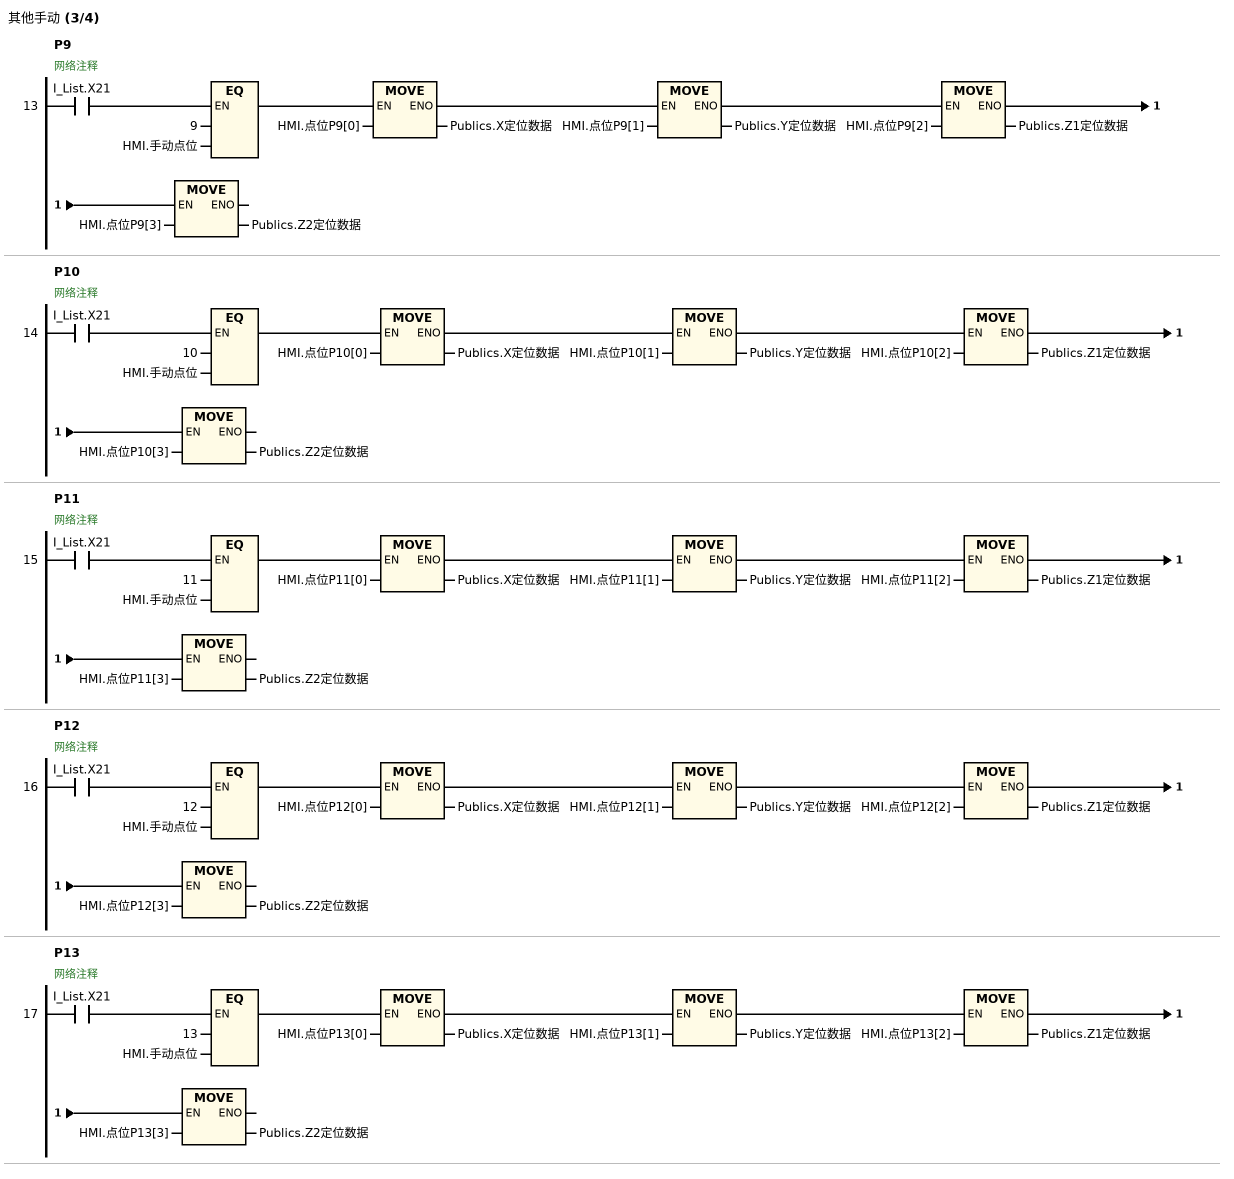
// NETWORK 13: P9
// 网络注释
_w9 := I_List.X21 AND 9 = HMI.手动点位;
IF _w9 THEN Publics.X定位数据 := HMI.点位P9[0]; END_IF
IF _w9 THEN Publics.Y定位数据 := HMI.点位P9[1]; END_IF
IF _w9 THEN Publics.Z1定位数据 := HMI.点位P9[2]; END_IF
IF _w9 THEN Publics.Z2定位数据 := HMI.点位P9[3]; END_IF

// NETWORK 14: P10
// 网络注释
_w10 := I_List.X21 AND 10 = HMI.手动点位;
IF _w10 THEN Publics.X定位数据 := HMI.点位P10[0]; END_IF
IF _w10 THEN Publics.Y定位数据 := HMI.点位P10[1]; END_IF
IF _w10 THEN Publics.Z1定位数据 := HMI.点位P10[2]; END_IF
IF _w10 THEN Publics.Z2定位数据 := HMI.点位P10[3]; END_IF

// NETWORK 15: P11
// 网络注释
_w11 := I_List.X21 AND 11 = HMI.手动点位;
IF _w11 THEN Publics.X定位数据 := HMI.点位P11[0]; END_IF
IF _w11 THEN Publics.Y定位数据 := HMI.点位P11[1]; END_IF
IF _w11 THEN Publics.Z1定位数据 := HMI.点位P11[2]; END_IF
IF _w11 THEN Publics.Z2定位数据 := HMI.点位P11[3]; END_IF

// NETWORK 16: P12
// 网络注释
_w12 := I_List.X21 AND 12 = HMI.手动点位;
IF _w12 THEN Publics.X定位数据 := HMI.点位P12[0]; END_IF
IF _w12 THEN Publics.Y定位数据 := HMI.点位P12[1]; END_IF
IF _w12 THEN Publics.Z1定位数据 := HMI.点位P12[2]; END_IF
IF _w12 THEN Publics.Z2定位数据 := HMI.点位P12[3]; END_IF

// NETWORK 17: P13
// 网络注释
_w13 := I_List.X21 AND 13 = HMI.手动点位;
IF _w13 THEN Publics.X定位数据 := HMI.点位P13[0]; END_IF
IF _w13 THEN Publics.Y定位数据 := HMI.点位P13[1]; END_IF
IF _w13 THEN Publics.Z1定位数据 := HMI.点位P13[2]; END_IF
IF _w13 THEN Publics.Z2定位数据 := HMI.点位P13[3]; END_IF

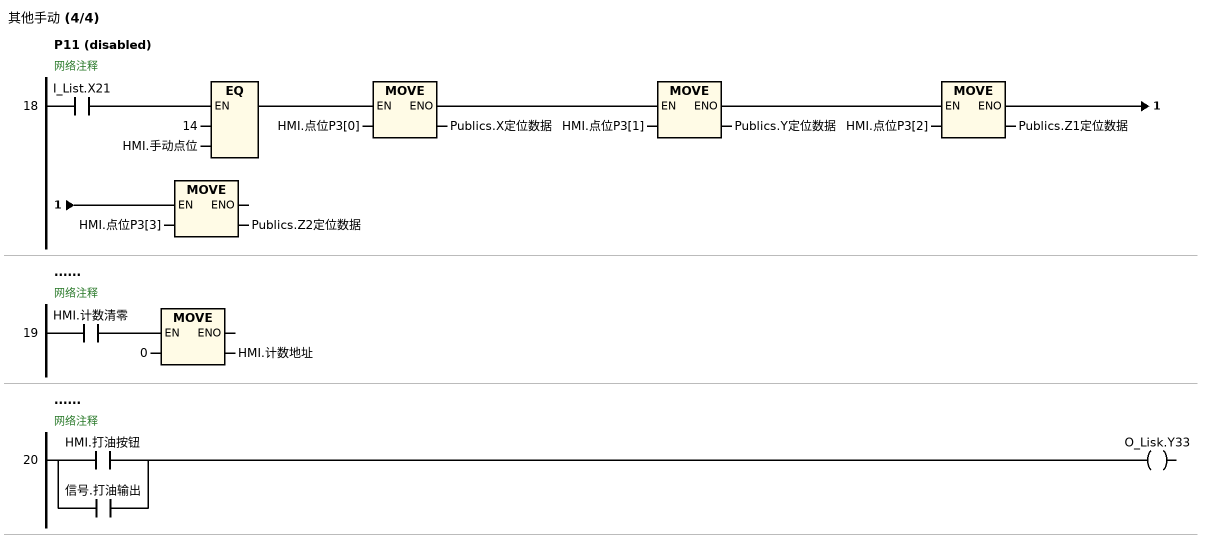
// NETWORK 18: P11 (disabled)
// 网络注释
// _w14 := I_List.X21 AND 14 = HMI.手动点位;
// IF _w14 THEN Publics.X定位数据 := HMI.点位P3[0]; END_IF
// IF _w14 THEN Publics.Y定位数据 := HMI.点位P3[1]; END_IF
// IF _w14 THEN Publics.Z1定位数据 := HMI.点位P3[2]; END_IF
// IF _w14 THEN Publics.Z2定位数据 := HMI.点位P3[3]; END_IF

// NETWORK 19: ......
// 网络注释
IF HMI.计数清零 THEN HMI.计数地址 := 0; END_IF

// NETWORK 20: ......
// 网络注释
O_Lisk.Y33 := HMI.打油按钮 OR 信号.打油输出;

END_PROGRAM

// Device/Application/Servo_Ctrol
PROGRAM Servo_Ctrol
VAR
	总线复位: BOOL;
	SMC3_ReinitDrive_0: SMC3_ReinitDrive;
	SMC3_ReinitDrive_1: SMC3_ReinitDrive;
	SMC3_ReinitDrive_2: SMC3_ReinitDrive;
	SMC3_ReinitDrive_3: SMC3_ReinitDrive;
	Y轴_使能: MC_Power;
	Z2轴_使能: MC_Power;
	Z1轴_使能: MC_Power;
	X轴_使能: MC_Power;
	MC_Jog_0: MC_Jog;
	Y轴_JOG: MC_Jog;
	Z2轴_JOG: MC_Jog;
	Z1轴_JOG: MC_Jog;
	X轴_JOG: MC_Jog;
	AXIS3: AXIS_REF_SM3;
	MC_Reset_0: MC_Reset;
	MC_Reset_1: MC_Reset;
	MC_Reset_2: MC_Reset;
	MC_Reset_3: MC_Reset;
	MC_ReadStatus_0: MC_ReadStatus;
	MC_ReadAxisError_0: MC_ReadAxisError;
	MC_ReadActualPosition_0: MC_ReadActualPosition;
	MC_ReadActualPosition_1: MC_ReadActualPosition;
	MC_ReadActualPosition_2: MC_ReadActualPosition;
	MC_ReadActualPosition_3: MC_ReadActualPosition;
	MC_Halt_0: MC_Halt;
	MC_Halt_1: MC_Halt;
	MC_Halt_2: MC_Halt;
	MC_Halt_3: MC_Halt;
	MC_Stop_0: MC_Stop;
	MC_Stop_1: MC_Stop;
	MC_Stop_2: MC_Stop;
	MC_Stop_3: MC_Stop;
	Z2定位: MC_MoveAbsolute;
	Z1定位: MC_MoveAbsolute;
	Y定位: MC_MoveAbsolute;
	X定位: MC_MoveAbsolute;
	MC_Home_0: MC_Home;
	MC_Home_1: MC_Home;
	MC_Home_2: MC_Home;
	MC_Home_3: MC_Home;
	ALM0: BOOL;
	ALM1: BOOL;
	ALM2: BOOL;
	ALM3: BOOL;
END_VAR
VAR // added by the converter: edge detectors and wires of the graphical bodies
    _rt1, _rt2, _rt3, _rt4, _rt5, _rt6, _rt7 : R_TRIG;
END_VAR

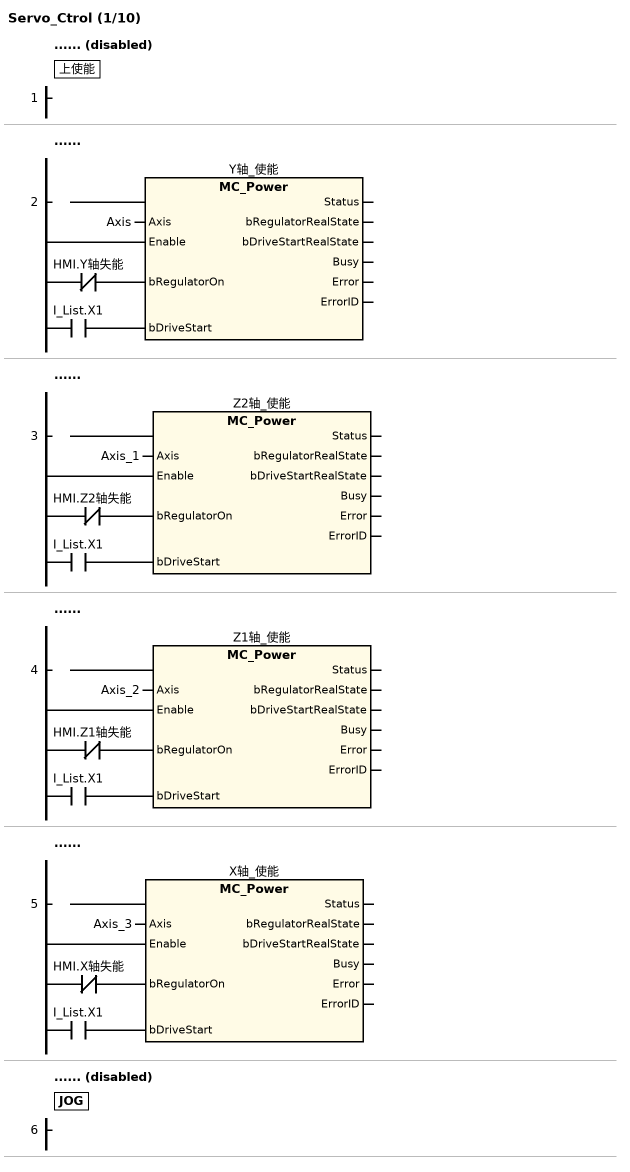
// NETWORK 1: ...... (disabled)
// label: 上使能

// NETWORK 2: ......
Y轴_使能(Axis := Axis, Enable := TRUE, bRegulatorOn := NOT HMI.Y轴失能, bDriveStart := I_List.X1); // MC_Power

// NETWORK 3: ......
Z2轴_使能(Axis := Axis_1, Enable := TRUE, bRegulatorOn := NOT HMI.Z2轴失能, bDriveStart := I_List.X1); // MC_Power

// NETWORK 4: ......
Z1轴_使能(Axis := Axis_2, Enable := TRUE, bRegulatorOn := NOT HMI.Z1轴失能, bDriveStart := I_List.X1); // MC_Power

// NETWORK 5: ......
X轴_使能(Axis := Axis_3, Enable := TRUE, bRegulatorOn := NOT HMI.X轴失能, bDriveStart := I_List.X1); // MC_Power

// NETWORK 6: ...... (disabled)
// label: JOG

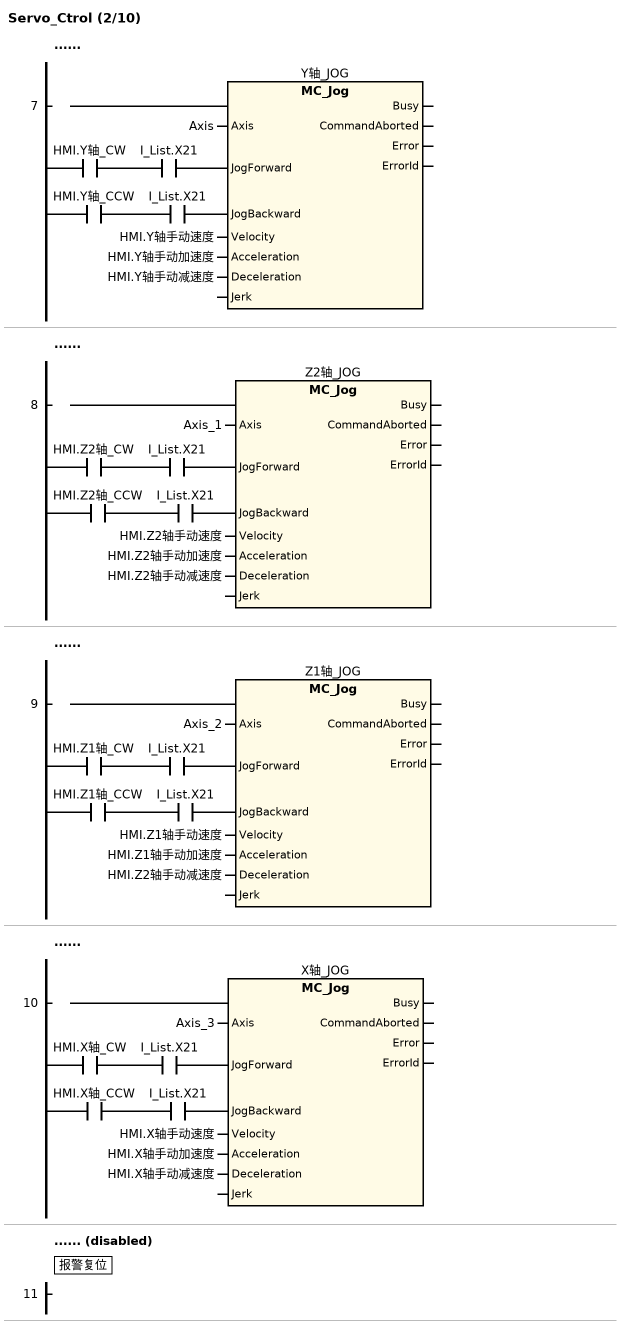
// NETWORK 7: ......
Y轴_JOG(
    Axis := Axis,
    JogForward := HMI.Y轴_CW AND I_List.X21,
    JogBackward := HMI.Y轴_CCW AND I_List.X21,
    Velocity := HMI.Y轴手动速度,
    Acceleration := HMI.Y轴手动加速度,
    Deceleration := HMI.Y轴手动减速度); // MC_Jog

// NETWORK 8: ......
Z2轴_JOG(
    Axis := Axis_1,
    JogForward := HMI.Z2轴_CW AND I_List.X21,
    JogBackward := HMI.Z2轴_CCW AND I_List.X21,
    Velocity := HMI.Z2轴手动速度,
    Acceleration := HMI.Z2轴手动加速度,
    Deceleration := HMI.Z2轴手动减速度); // MC_Jog

// NETWORK 9: ......
Z1轴_JOG(
    Axis := Axis_2,
    JogForward := HMI.Z1轴_CW AND I_List.X21,
    JogBackward := HMI.Z1轴_CCW AND I_List.X21,
    Velocity := HMI.Z1轴手动速度,
    Acceleration := HMI.Z1轴手动加速度,
    Deceleration := HMI.Z2轴手动减速度); // MC_Jog

// NETWORK 10: ......
X轴_JOG(
    Axis := Axis_3,
    JogForward := HMI.X轴_CW AND I_List.X21,
    JogBackward := HMI.X轴_CCW AND I_List.X21,
    Velocity := HMI.X轴手动速度,
    Acceleration := HMI.X轴手动加速度,
    Deceleration := HMI.X轴手动减速度); // MC_Jog

// NETWORK 11: ...... (disabled)
// label: 报警复位

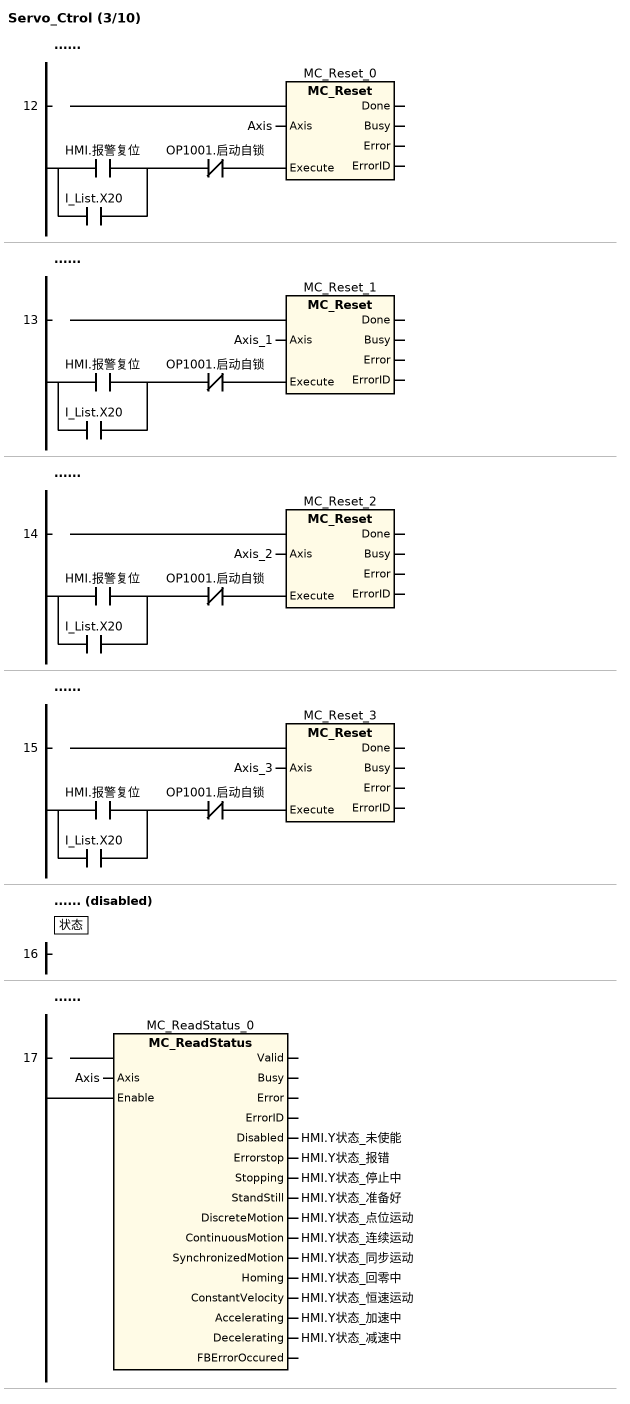
// NETWORK 12: ......
MC_Reset_0(Axis := Axis, Execute := (HMI.报警复位 OR I_List.X20) AND NOT OP1001.启动自锁); // MC_Reset

// NETWORK 13: ......
MC_Reset_1(Axis := Axis_1, Execute := (HMI.报警复位 OR I_List.X20) AND NOT OP1001.启动自锁); // MC_Reset

// NETWORK 14: ......
MC_Reset_2(Axis := Axis_2, Execute := (HMI.报警复位 OR I_List.X20) AND NOT OP1001.启动自锁); // MC_Reset

// NETWORK 15: ......
MC_Reset_3(Axis := Axis_3, Execute := (HMI.报警复位 OR I_List.X20) AND NOT OP1001.启动自锁); // MC_Reset

// NETWORK 16: ...... (disabled)
// label: 状态

// NETWORK 17: ......
MC_ReadStatus_0(
    Axis := Axis,
    Enable := TRUE,
    Disabled => HMI.Y状态_未使能,
    Errorstop => HMI.Y状态_报错,
    Stopping => HMI.Y状态_停止中,
    StandStill => HMI.Y状态_准备好,
    DiscreteMotion => HMI.Y状态_点位运动,
    ContinuousMotion => HMI.Y状态_连续运动,
    SynchronizedMotion => HMI.Y状态_同步运动,
    Homing => HMI.Y状态_回零中,
    ConstantVelocity => HMI.Y状态_恒速运动,
    Accelerating => HMI.Y状态_加速中,
    Decelerating => HMI.Y状态_减速中); // MC_ReadStatus

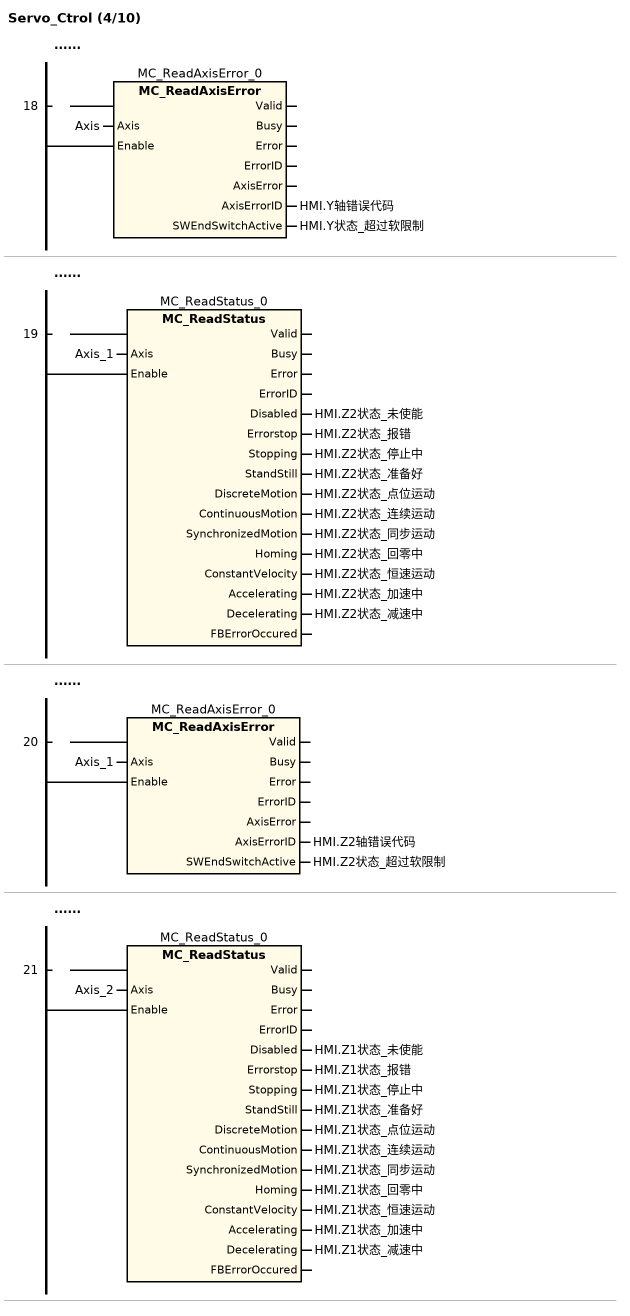
// NETWORK 18: ......
MC_ReadAxisError_0(
    Axis := Axis,
    Enable := TRUE,
    AxisErrorID => HMI.Y轴错误代码,
    SWEndSwitchActive => HMI.Y状态_超过软限制); // MC_ReadAxisError

// NETWORK 19: ......
MC_ReadStatus_0(
    Axis := Axis_1,
    Enable := TRUE,
    Disabled => HMI.Z2状态_未使能,
    Errorstop => HMI.Z2状态_报错,
    Stopping => HMI.Z2状态_停止中,
    StandStill => HMI.Z2状态_准备好,
    DiscreteMotion => HMI.Z2状态_点位运动,
    ContinuousMotion => HMI.Z2状态_连续运动,
    SynchronizedMotion => HMI.Z2状态_同步运动,
    Homing => HMI.Z2状态_回零中,
    ConstantVelocity => HMI.Z2状态_恒速运动,
    Accelerating => HMI.Z2状态_加速中,
    Decelerating => HMI.Z2状态_减速中); // MC_ReadStatus

// NETWORK 20: ......
MC_ReadAxisError_0(
    Axis := Axis_1,
    Enable := TRUE,
    AxisErrorID => HMI.Z2轴错误代码,
    SWEndSwitchActive => HMI.Z2状态_超过软限制); // MC_ReadAxisError

// NETWORK 21: ......
MC_ReadStatus_0(
    Axis := Axis_2,
    Enable := TRUE,
    Disabled => HMI.Z1状态_未使能,
    Errorstop => HMI.Z1状态_报错,
    Stopping => HMI.Z1状态_停止中,
    StandStill => HMI.Z1状态_准备好,
    DiscreteMotion => HMI.Z1状态_点位运动,
    ContinuousMotion => HMI.Z1状态_连续运动,
    SynchronizedMotion => HMI.Z1状态_同步运动,
    Homing => HMI.Z1状态_回零中,
    ConstantVelocity => HMI.Z1状态_恒速运动,
    Accelerating => HMI.Z1状态_加速中,
    Decelerating => HMI.Z1状态_减速中); // MC_ReadStatus

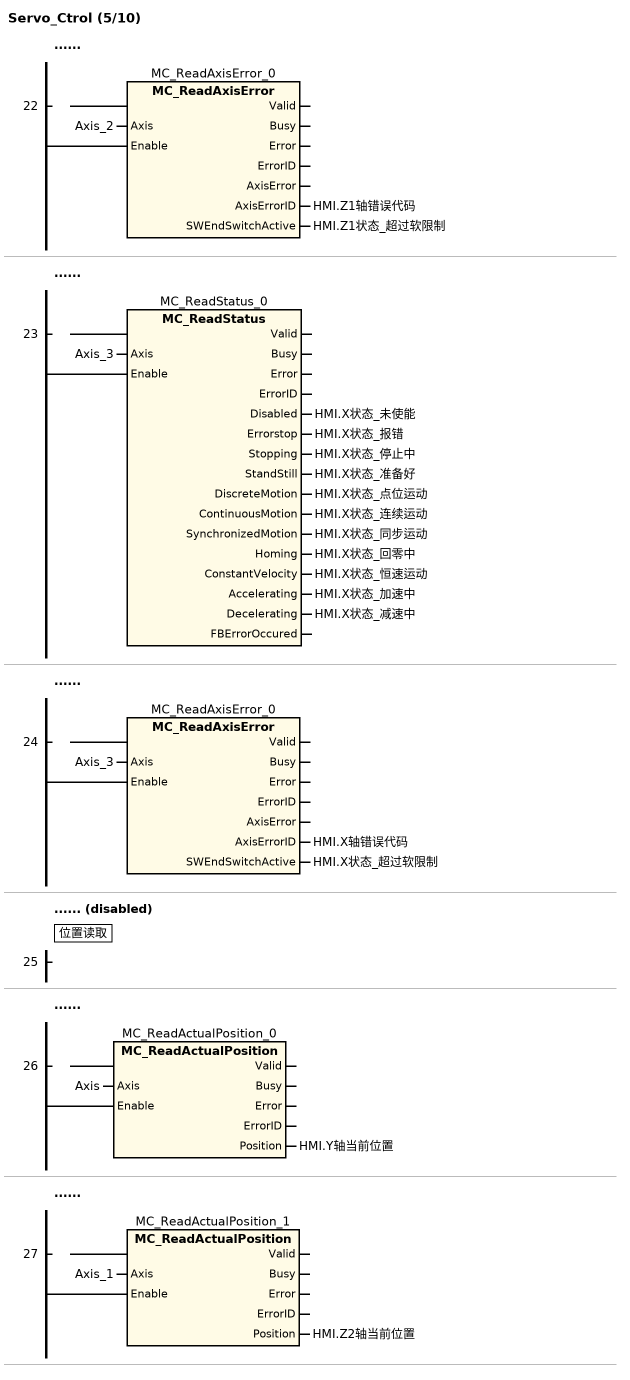
// NETWORK 22: ......
MC_ReadAxisError_0(
    Axis := Axis_2,
    Enable := TRUE,
    AxisErrorID => HMI.Z1轴错误代码,
    SWEndSwitchActive => HMI.Z1状态_超过软限制); // MC_ReadAxisError

// NETWORK 23: ......
MC_ReadStatus_0(
    Axis := Axis_3,
    Enable := TRUE,
    Disabled => HMI.X状态_未使能,
    Errorstop => HMI.X状态_报错,
    Stopping => HMI.X状态_停止中,
    StandStill => HMI.X状态_准备好,
    DiscreteMotion => HMI.X状态_点位运动,
    ContinuousMotion => HMI.X状态_连续运动,
    SynchronizedMotion => HMI.X状态_同步运动,
    Homing => HMI.X状态_回零中,
    ConstantVelocity => HMI.X状态_恒速运动,
    Accelerating => HMI.X状态_加速中,
    Decelerating => HMI.X状态_减速中); // MC_ReadStatus

// NETWORK 24: ......
MC_ReadAxisError_0(
    Axis := Axis_3,
    Enable := TRUE,
    AxisErrorID => HMI.X轴错误代码,
    SWEndSwitchActive => HMI.X状态_超过软限制); // MC_ReadAxisError

// NETWORK 25: ...... (disabled)
// label: 位置读取

// NETWORK 26: ......
MC_ReadActualPosition_0(Axis := Axis, Enable := TRUE, Position => HMI.Y轴当前位置); // MC_ReadActualPosition

// NETWORK 27: ......
MC_ReadActualPosition_1(Axis := Axis_1, Enable := TRUE, Position => HMI.Z2轴当前位置); // MC_ReadActualPosition

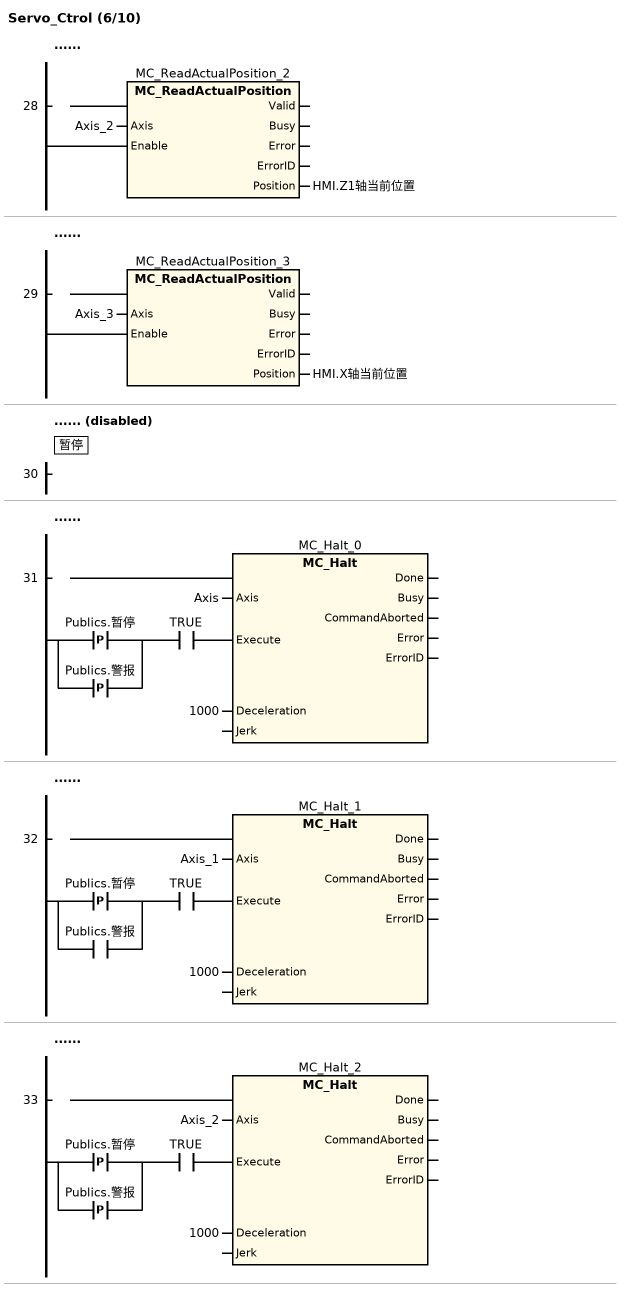
// NETWORK 28: ......
MC_ReadActualPosition_2(Axis := Axis_2, Enable := TRUE, Position => HMI.Z1轴当前位置); // MC_ReadActualPosition

// NETWORK 29: ......
MC_ReadActualPosition_3(Axis := Axis_3, Enable := TRUE, Position => HMI.X轴当前位置); // MC_ReadActualPosition

// NETWORK 30: ...... (disabled)
// label: 暂停

// NETWORK 31: ......
_rt1(CLK := Publics.暂停);
_rt2(CLK := Publics.警报);
MC_Halt_0(Axis := Axis, Execute := (_rt1.Q OR _rt2.Q) AND TRUE, Deceleration := 1000); // MC_Halt

// NETWORK 32: ......
_rt3(CLK := Publics.暂停);
MC_Halt_1(Axis := Axis_1, Execute := (_rt3.Q OR Publics.警报) AND TRUE, Deceleration := 1000); // MC_Halt

// NETWORK 33: ......
_rt4(CLK := Publics.暂停);
_rt5(CLK := Publics.警报);
MC_Halt_2(Axis := Axis_2, Execute := (_rt4.Q OR _rt5.Q) AND TRUE, Deceleration := 1000); // MC_Halt

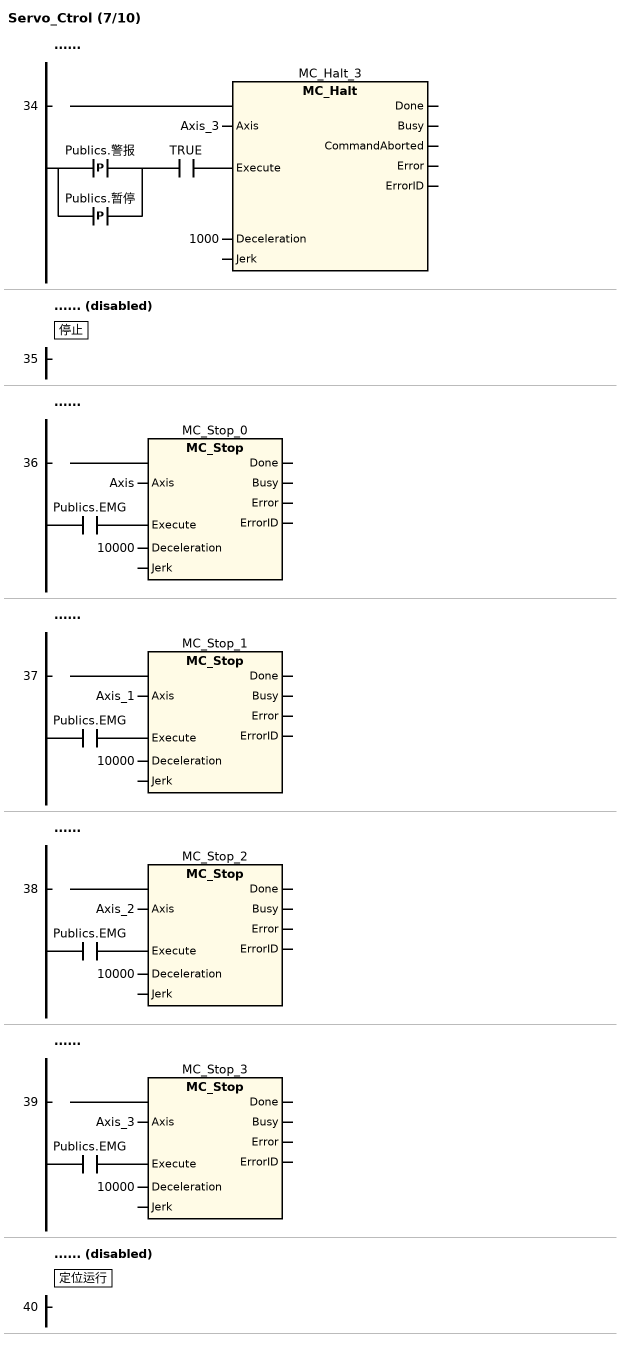
// NETWORK 34: ......
_rt6(CLK := Publics.警报);
_rt7(CLK := Publics.暂停);
MC_Halt_3(Axis := Axis_3, Execute := (_rt6.Q OR _rt7.Q) AND TRUE, Deceleration := 1000); // MC_Halt

// NETWORK 35: ...... (disabled)
// label: 停止

// NETWORK 36: ......
MC_Stop_0(Axis := Axis, Execute := Publics.EMG, Deceleration := 10000); // MC_Stop

// NETWORK 37: ......
MC_Stop_1(Axis := Axis_1, Execute := Publics.EMG, Deceleration := 10000); // MC_Stop

// NETWORK 38: ......
MC_Stop_2(Axis := Axis_2, Execute := Publics.EMG, Deceleration := 10000); // MC_Stop

// NETWORK 39: ......
MC_Stop_3(Axis := Axis_3, Execute := Publics.EMG, Deceleration := 10000); // MC_Stop

// NETWORK 40: ...... (disabled)
// label: 定位运行

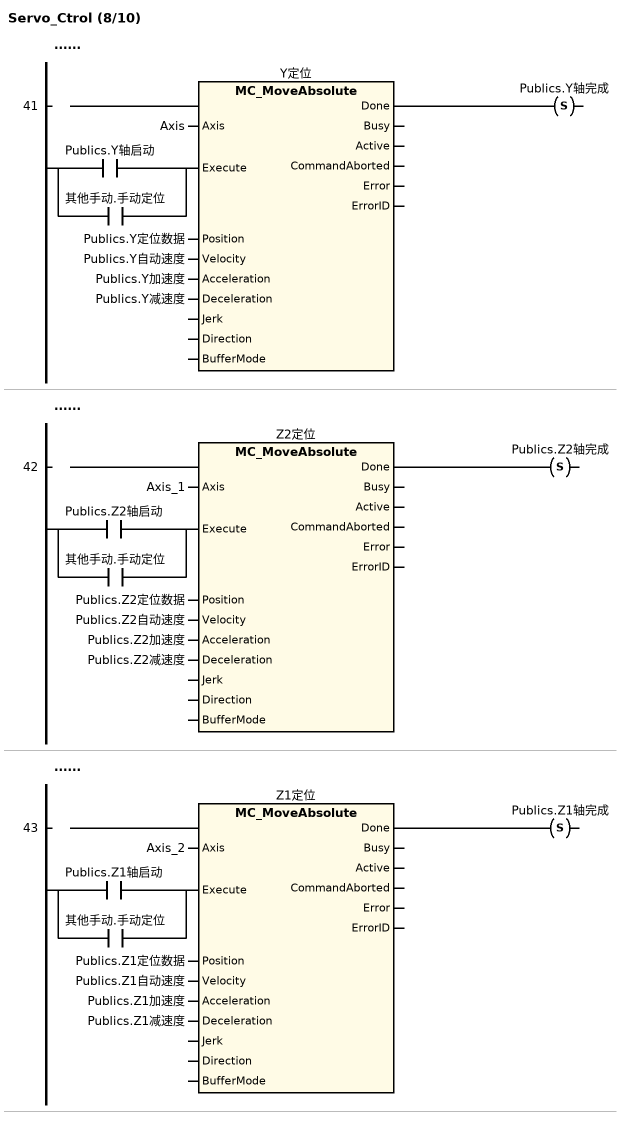
// NETWORK 41: ......
Y定位(
    Axis := Axis,
    Execute := Publics.Y轴启动 OR 其他手动.手动定位,
    Position := Publics.Y定位数据,
    Velocity := Publics.Y自动速度,
    Acceleration := Publics.Y加速度,
    Deceleration := Publics.Y减速度); // MC_MoveAbsolute
Publics.Y轴完成 S= Y定位.Done;

// NETWORK 42: ......
Z2定位(
    Axis := Axis_1,
    Execute := Publics.Z2轴启动 OR 其他手动.手动定位,
    Position := Publics.Z2定位数据,
    Velocity := Publics.Z2自动速度,
    Acceleration := Publics.Z2加速度,
    Deceleration := Publics.Z2减速度); // MC_MoveAbsolute
Publics.Z2轴完成 S= Z2定位.Done;

// NETWORK 43: ......
Z1定位(
    Axis := Axis_2,
    Execute := Publics.Z1轴启动 OR 其他手动.手动定位,
    Position := Publics.Z1定位数据,
    Velocity := Publics.Z1自动速度,
    Acceleration := Publics.Z1加速度,
    Deceleration := Publics.Z1减速度); // MC_MoveAbsolute
Publics.Z1轴完成 S= Z1定位.Done;

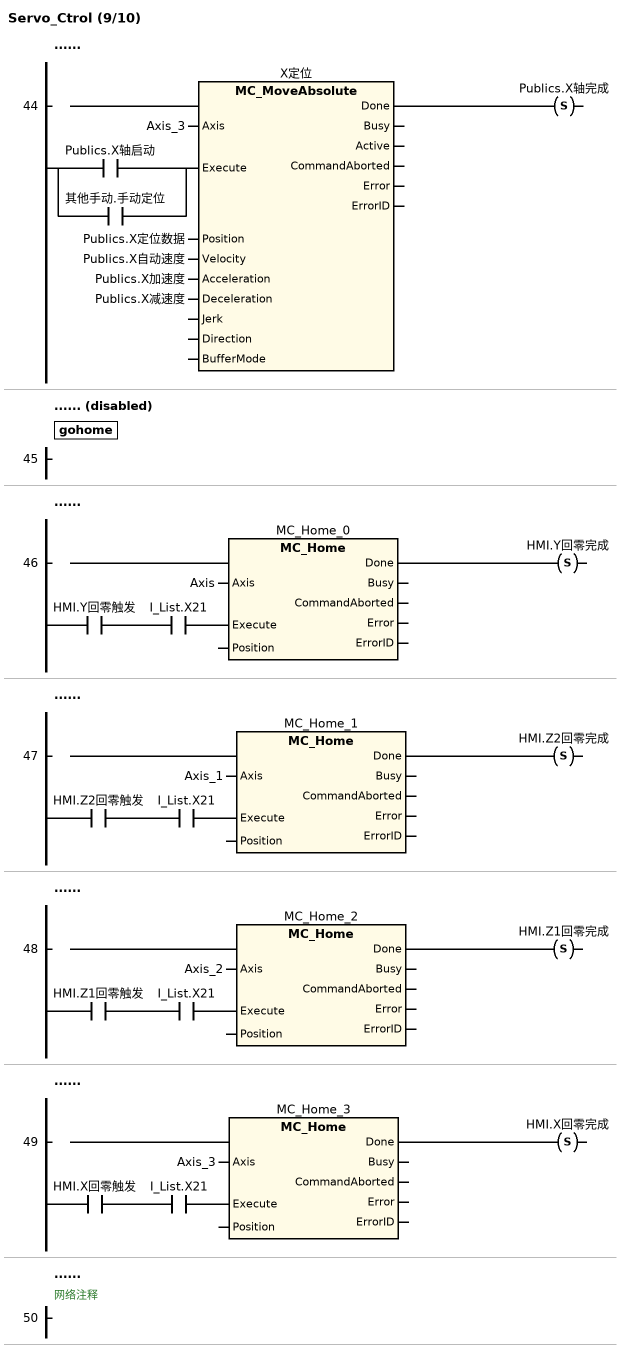
// NETWORK 44: ......
X定位(
    Axis := Axis_3,
    Execute := Publics.X轴启动 OR 其他手动.手动定位,
    Position := Publics.X定位数据,
    Velocity := Publics.X自动速度,
    Acceleration := Publics.X加速度,
    Deceleration := Publics.X减速度); // MC_MoveAbsolute
Publics.X轴完成 S= X定位.Done;

// NETWORK 45: ...... (disabled)
// label: gohome

// NETWORK 46: ......
MC_Home_0(Axis := Axis, Execute := HMI.Y回零触发 AND I_List.X21); // MC_Home
HMI.Y回零完成 S= MC_Home_0.Done;

// NETWORK 47: ......
MC_Home_1(Axis := Axis_1, Execute := HMI.Z2回零触发 AND I_List.X21); // MC_Home
HMI.Z2回零完成 S= MC_Home_1.Done;

// NETWORK 48: ......
MC_Home_2(Axis := Axis_2, Execute := HMI.Z1回零触发 AND I_List.X21); // MC_Home
HMI.Z1回零完成 S= MC_Home_2.Done;

// NETWORK 49: ......
MC_Home_3(Axis := Axis_3, Execute := HMI.X回零触发 AND I_List.X21); // MC_Home
HMI.X回零完成 S= MC_Home_3.Done;

// NETWORK 50: ......
// 网络注释

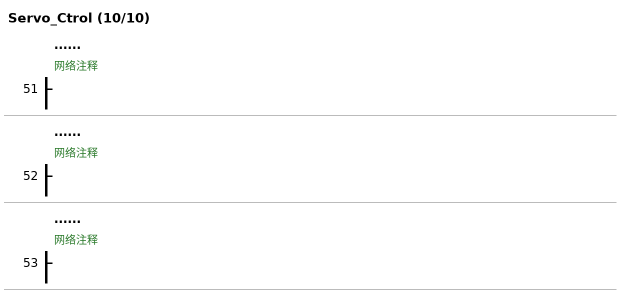
// NETWORK 51: ......
// 网络注释

// NETWORK 52: ......
// 网络注释

// NETWORK 53: ......
// 网络注释

END_PROGRAM

// Device/Application/ITF
INTERFACE ITF

END_INTERFACE

// Device/Application/FunctionBlock/FB_CylinderDouble
FUNCTION_BLOCK FB_CylinderDouble
VAR_IN_OUT
	///气缸控制、状态和报警
	stCylvar: CYLINDER_REF;
END_VAR
VAR_INPUT
	///安全条件
	xReady: BOOL;
	///报警复位
	xReset: BOOL;
	///手动控制,每on一次,则反转输出点状态
	xManuCmd: BOOL;
	///原位检测
	xBackSensor: BOOL;
	///到位检测
	xFrontSensor: BOOL;
	///手自动不一致报警无效
	xManuAlmDisable: BOOL;
	///原位检测无效
	xBackSensorDisable: BOOL;
	///到位检测无效	
	xFrontSensorDisable: BOOL;
	///原位延时	
	wBackDelay: WORD;
	///到位延时
	wFrontDelay: WORD;
END_VAR
VAR_OUTPUT
	///输出点,对应双控气缸原位电磁阀
	xOutputA: BOOL;
	///输出点,应双控气缸到位电磁阀
	xOutputB: BOOL;
	///未满足安全条件报警
	f_xNotRdyAlm: BOOL;
	///手自动不一致报警	
	f_xManuAlm: BOOL;
	///未在原位报警
	f_xBackAlm: BOOL;
	///未到位报警	
	f_xFrontAlm: BOOL;
	///气缸处于不受控制状态报警
	f_xUncontrolledAlm: BOOL;
END_VAR
VAR
	///获取自动控制的上升沿
	fbAutoRise: R_TRIG;
	///获取自动控制的下升沿
	fbAutoFall: F_TRIG;
	///获取手动控制的下升沿
	fbManuFall: F_TRIG;
	///获取复位信号的上升沿
	fbResetRise: R_TRIG;
	///原位状态延时,用于输出原位状态
	fbBackTon: TON;
	///到位状态延时,用于输出到位状态	
	fbFrontTon: TON;
	///获取原位状态下降沿
	fbBackFall: F_TRIG;
	///获取到位状态下降沿
	fbFrontFall: F_TRIG;
	///原位动作超时,用于输出未在原位位置报警
	fbBackWait: TON;
	///到位动作超时,用于输出未在原位位置报警
	fbFrontWait: TON;
END_VAR

   //初始化时返回原位
   IF  xReady AND stCylvar.xInit AND ( NOT xManuCmd ) THEN
	     xOutputA  := TRUE; 
         xOutputB  := FALSE;
		 f_xManuAlm  := FALSE;
		 stCylvar.xInit  := FALSE;	  	  	 	  
   END_IF	  
   
   //获取手动控制、自动控制的边沿信号
   fbManuFall(CLK:=xManuCmd , Q=> );
   fbAutoRise(CLK:=stCylvar.xAutoCmd , Q=> );
   fbAutoFall(CLK:=stCylvar.xAutoCmd , Q=> );
   
   //1,手动操作时，如果满足安全条件且未屏蔽手自动不一致报警时，则输出点A反转，输出点B取输出点A的反逻辑
   IF xReady AND (NOT xManuAlmDisable) AND fbManuFall.Q THEN
	   xOutputA  := NOT xOutputA; 
	   xOutputB  := NOT xOutputA;
	   
	//手动操作生效时，判断输出点状态与自动命令是否一致，不一致时,置位手动操作执行中报警；一致时复位该报警。
	//当因安全条件不满足导致自动命令未执行时，可通过手动操作控制其动作执行,此时手动操作并不引起手动操作执行中报警。
   	   IF (stCylvar.xAutoCmd AND (NOT xManuAlmDisable) ) XOR xOutputB THEN
   	   	    f_xManuAlm  :=TRUE;
   	   ELSE 
   	   	    f_xManuAlm  :=FALSE;
   	   END_IF
   END_IF
   //2,手动操作时，如果满足安全条件且屏蔽了手自动不一致报警时，则自动控制点反转、复位手自动不一致报警，  
    IF xReady AND  xManuAlmDisable AND fbManuFall.Q THEN
   	    stCylvar.xAutoCmd  := NOT stCylvar.xAutoCmd ;
		f_xManuAlm  :=FALSE;		  	 	
    END_IF
   
   //自动命令置位时，如满足安全条件，则输出点A复位、 输出点B置位。
   IF xReady AND fbAutoRise.Q THEN
   	    xOutputA  :=FALSE;
		xOutputB  :=TRUE;
		
   END_IF
   //自动命令复位时，如满足安全条件，则输出点A置位、 输出点B复位。
   IF xReady AND fbAutoFall.Q THEN
   	    xOutputA  :=TRUE;
		xOutputB  :=FALSE;		
   END_IF
   
   
   //到位状态输出
   fbFrontTon(IN:=( NOT xOutputA ) AND xOutputB AND ( xFrontSensor OR xFrontSensorDisable ) AND ( NOT xBackSensor ) , PT:= WORD_TO_TIME ( wFrontDelay *10 ), Q=> stCylvar.xIsFront, ET=> );
   
   //原位状态输出
   fbBackTon(IN:= xOutputA  AND ( NOT xOutputB) AND ( NOT xFrontSensor ) AND ( xBackSensor OR xBackSensorDisable ) , PT:= WORD_TO_TIME ( wBackDelay *10 ) , Q=> stCylvar.xIsBack, ET=> );
   
   
   //报警复位
   fbResetRise(CLK:= xReset, Q=> );
   IF fbResetRise.Q THEN
   	   f_xNotRdyAlm := FALSE;
	   f_xFrontAlm := FALSE;
	   f_xBackAlm := FALSE;
	   f_xUncontrolledAlm := FALSE;
   
   END_IF
   
   
   //未满足安全条件报警
   //当手动操作或自动命令状态发生改变时，如果不能满足安全条件，则输出未满足安全条件报警
   IF ( fbManuFall.Q OR fbAutoRise.Q OR fbAutoFall.Q ) AND ( NOT xReady ) THEN
   	   f_xNotRdyAlm := TRUE; 
   END_IF
   
   
   //未在原位报警
   //自动命令变OFF后(上电后气缸处于自由状态时不判断)，延时5秒，如果原位标志未变为ON、且未发生手动操作和安全条件报警，则输出未到原位报警
   fbBackWait(IN:= ( NOT stCylvar.xAutoCmd ) AND ( xOutputA OR xOutputB ) , PT:= T#5S , Q=> , ET=> );
   fbBackFall(CLK:= stCylvar.xIsBack , Q=> );
   IF (( fbBackWait.Q AND (NOT stCylvar.xIsBack )) OR (( NOT stCylvar.xAutoCmd ) AND fbBackFall.Q )) AND  ( NOT f_xManuAlm ) AND  ( NOT f_xNotRdyAlm ) THEN
   	    f_xBackAlm := TRUE;
   END_IF
   
   
   //未在到位报警
   //自动命令变ON后，延时5秒，如果到位标志未变为ON、且未发生手动操作和安全条件报警，则输出未到位报警
   fbFrontWait(IN:= stCylvar.xAutoCmd , PT:= T#5S , Q=> , ET=> );
   fbFrontFall(CLK:= stCylvar.xIsFront, Q=> );
   IF ( ( fbFrontWait.Q AND ( NOT stCylvar.xIsFront ) ) OR (stCylvar.xAutoCmd AND fbFrontFall.Q )) AND ( NOT f_xManuAlm ) AND ( NOT f_xNotRdyAlm ) THEN
   	    f_xFrontAlm := TRUE;   
   END_IF      
   
   
   //不受控状态报警
   IF NOT ( xOutputA OR xOutputB ) THEN
   	    f_xUncontrolledAlm := TRUE;
   END_IF

END_FUNCTION_BLOCK

// Device/Application/POU
PROGRAM POU
VAR
	当前步: uint;
	下一步: uint;
	定位位置: ARRAY[0..3] OF Lreal;
	LS_4AxisLine_0: LS_4AxisLine;
	避开扫描周期: BOOL;
	所有轴启动: BOOL;
	轴运行完成: BOOL;
END_VAR
VAR // added by the converter: edge detectors and wires of the graphical bodies
    _w1, _w2, _w3, _w4, _w5, _w6, _w7, _w8, _w9, _w10, _w11, _w12 : BOOL;
END_VAR

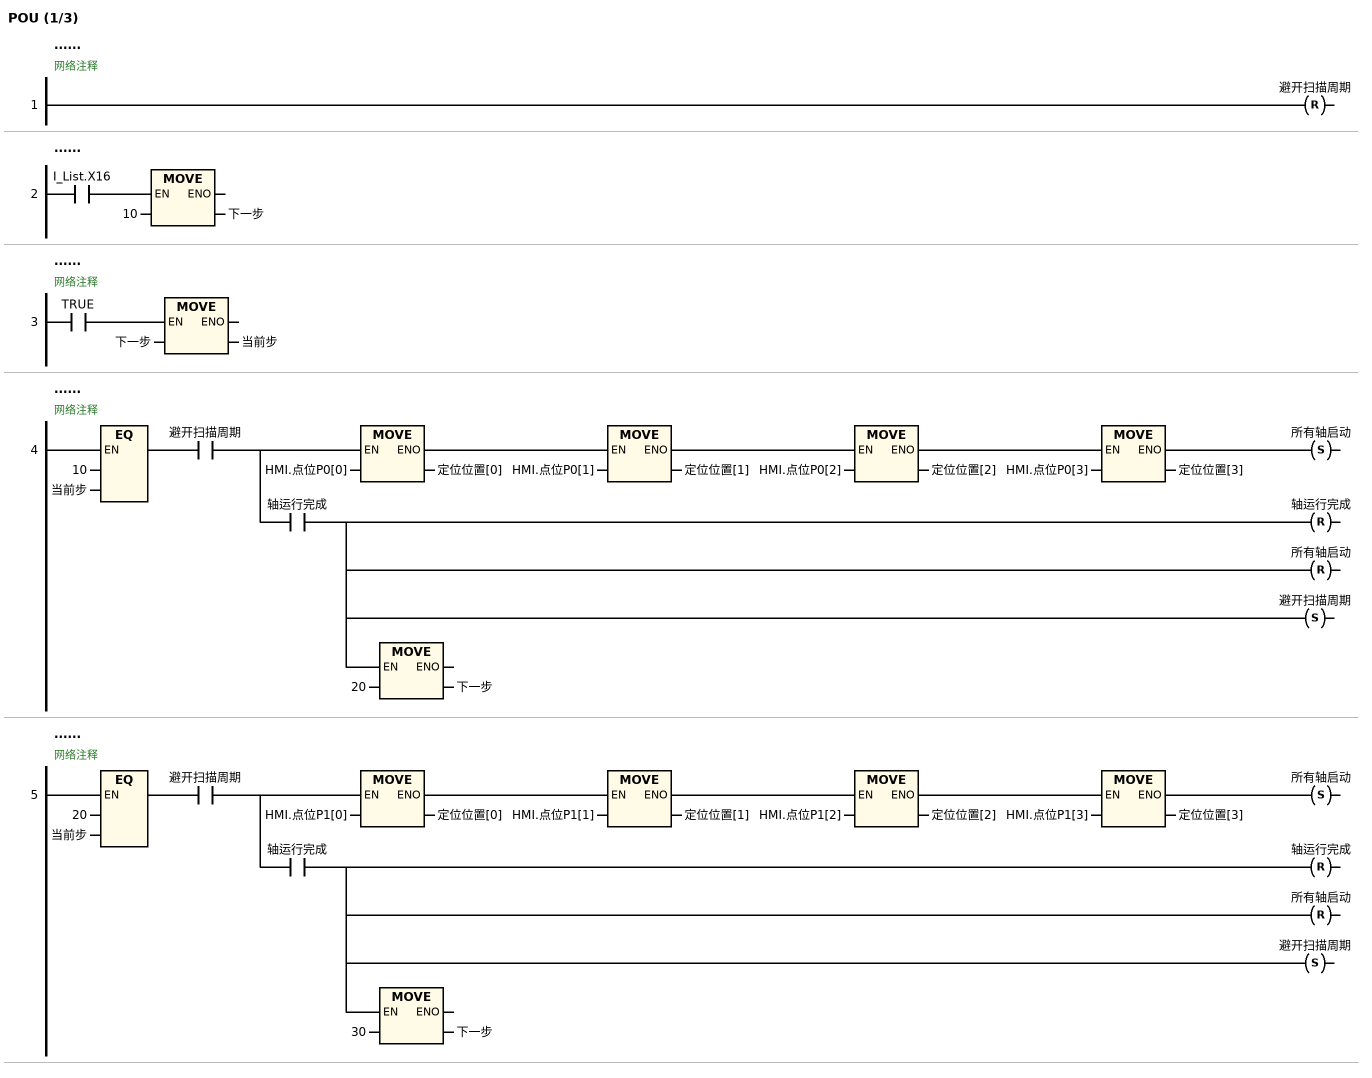
// NETWORK 1: ......
// 网络注释
避开扫描周期 R= TRUE;

// NETWORK 2: ......
IF I_List.X16 THEN 下一步 := 10; END_IF

// NETWORK 3: ......
// 网络注释
当前步 := 下一步;

// NETWORK 4: ......
// 网络注释
_w1 := 10 = 当前步 AND 避开扫描周期;
IF _w1 THEN 定位位置[0] := HMI.点位P0[0]; END_IF
IF _w1 THEN 定位位置[1] := HMI.点位P0[1]; END_IF
IF _w1 THEN 定位位置[2] := HMI.点位P0[2]; END_IF
IF _w1 THEN 定位位置[3] := HMI.点位P0[3]; END_IF
所有轴启动 S= _w1;
_w2 := _w1 AND 轴运行完成;
轴运行完成 R= _w2;
所有轴启动 R= _w2;
避开扫描周期 S= _w2;
IF _w2 THEN 下一步 := 20; END_IF

// NETWORK 5: ......
// 网络注释
_w3 := 20 = 当前步 AND 避开扫描周期;
IF _w3 THEN 定位位置[0] := HMI.点位P1[0]; END_IF
IF _w3 THEN 定位位置[1] := HMI.点位P1[1]; END_IF
IF _w3 THEN 定位位置[2] := HMI.点位P1[2]; END_IF
IF _w3 THEN 定位位置[3] := HMI.点位P1[3]; END_IF
所有轴启动 S= _w3;
_w4 := _w3 AND 轴运行完成;
轴运行完成 R= _w4;
所有轴启动 R= _w4;
避开扫描周期 S= _w4;
IF _w4 THEN 下一步 := 30; END_IF

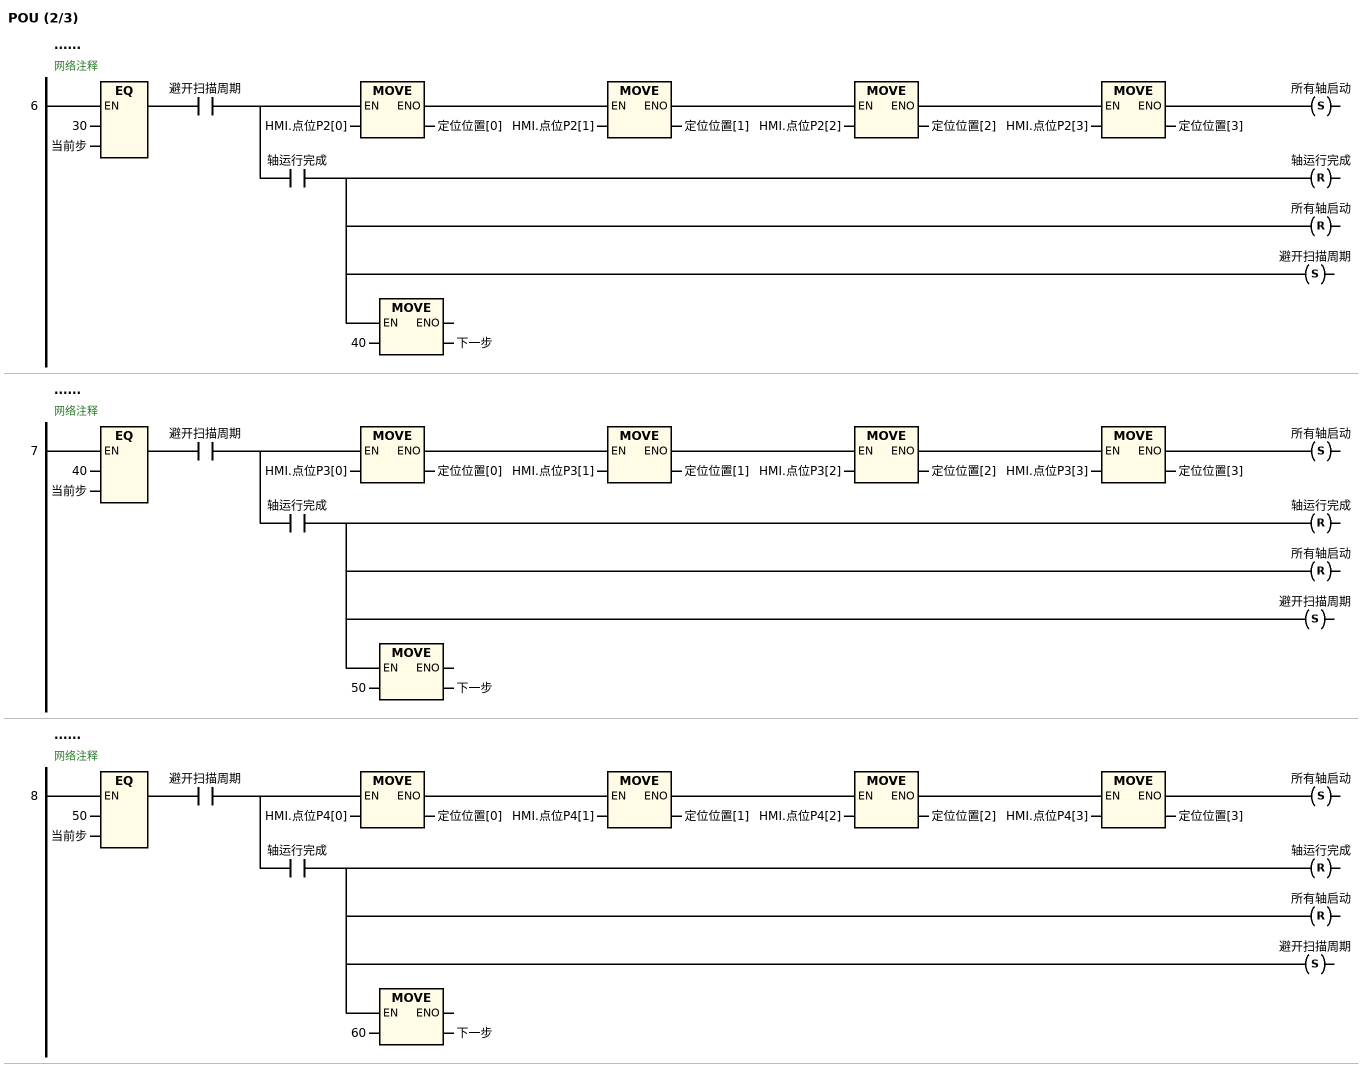
// NETWORK 6: ......
// 网络注释
_w5 := 30 = 当前步 AND 避开扫描周期;
IF _w5 THEN 定位位置[0] := HMI.点位P2[0]; END_IF
IF _w5 THEN 定位位置[1] := HMI.点位P2[1]; END_IF
IF _w5 THEN 定位位置[2] := HMI.点位P2[2]; END_IF
IF _w5 THEN 定位位置[3] := HMI.点位P2[3]; END_IF
所有轴启动 S= _w5;
_w6 := _w5 AND 轴运行完成;
轴运行完成 R= _w6;
所有轴启动 R= _w6;
避开扫描周期 S= _w6;
IF _w6 THEN 下一步 := 40; END_IF

// NETWORK 7: ......
// 网络注释
_w7 := 40 = 当前步 AND 避开扫描周期;
IF _w7 THEN 定位位置[0] := HMI.点位P3[0]; END_IF
IF _w7 THEN 定位位置[1] := HMI.点位P3[1]; END_IF
IF _w7 THEN 定位位置[2] := HMI.点位P3[2]; END_IF
IF _w7 THEN 定位位置[3] := HMI.点位P3[3]; END_IF
所有轴启动 S= _w7;
_w8 := _w7 AND 轴运行完成;
轴运行完成 R= _w8;
所有轴启动 R= _w8;
避开扫描周期 S= _w8;
IF _w8 THEN 下一步 := 50; END_IF

// NETWORK 8: ......
// 网络注释
_w9 := 50 = 当前步 AND 避开扫描周期;
IF _w9 THEN 定位位置[0] := HMI.点位P4[0]; END_IF
IF _w9 THEN 定位位置[1] := HMI.点位P4[1]; END_IF
IF _w9 THEN 定位位置[2] := HMI.点位P4[2]; END_IF
IF _w9 THEN 定位位置[3] := HMI.点位P4[3]; END_IF
所有轴启动 S= _w9;
_w10 := _w9 AND 轴运行完成;
轴运行完成 R= _w10;
所有轴启动 R= _w10;
避开扫描周期 S= _w10;
IF _w10 THEN 下一步 := 60; END_IF

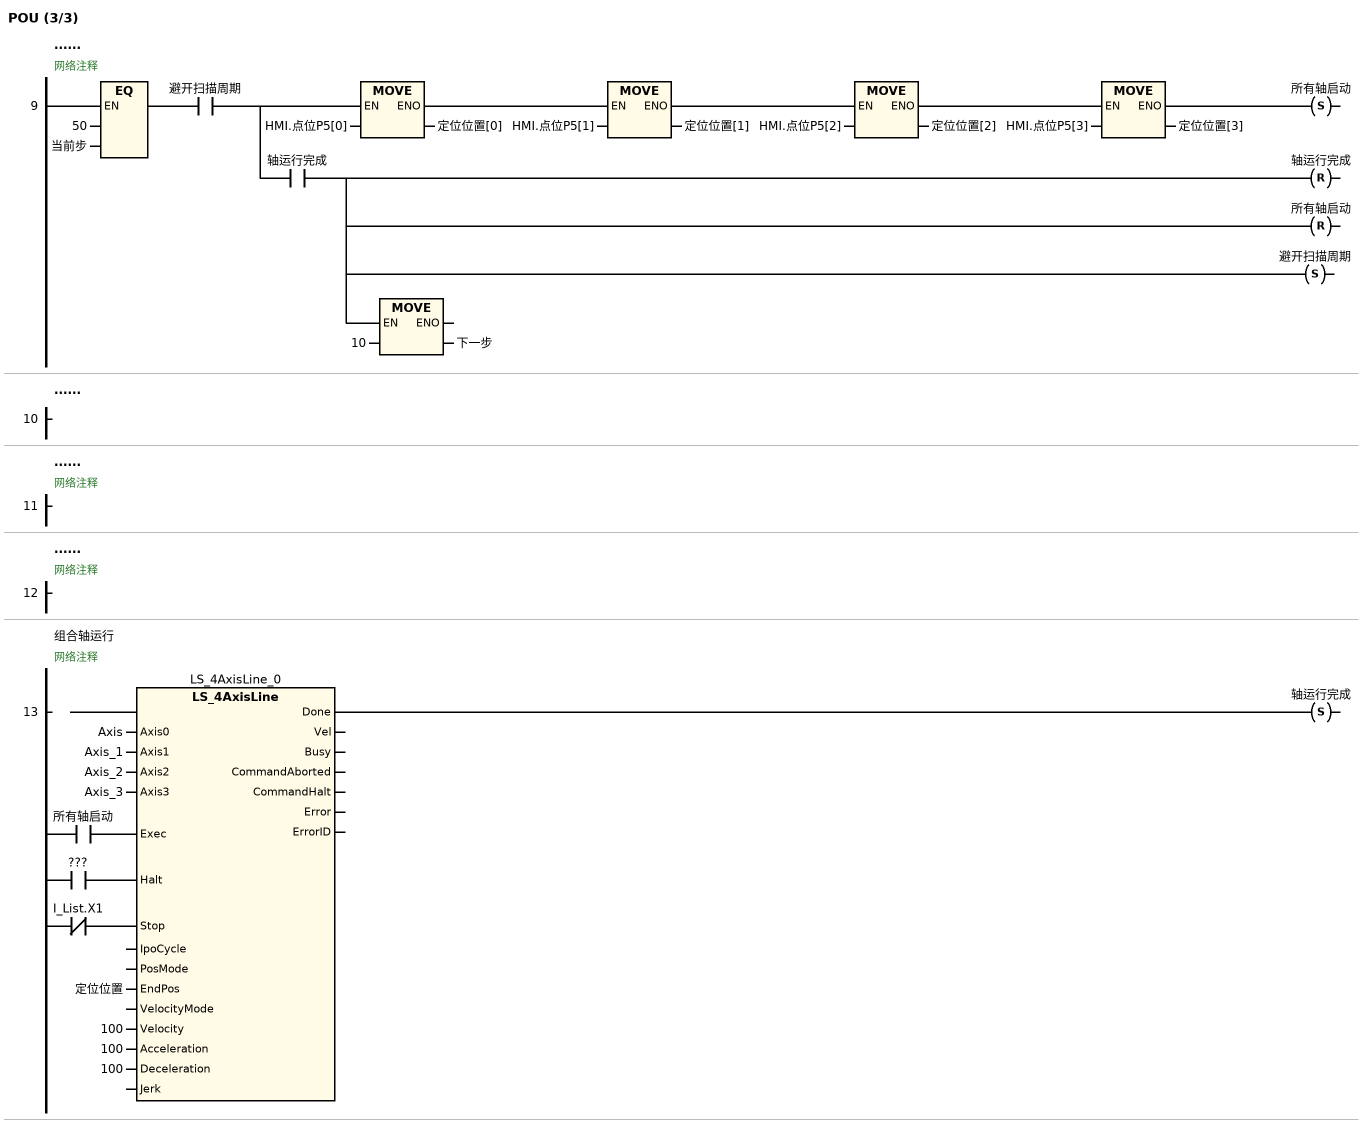
// NETWORK 9: ......
// 网络注释
_w11 := 50 = 当前步 AND 避开扫描周期;
IF _w11 THEN 定位位置[0] := HMI.点位P5[0]; END_IF
IF _w11 THEN 定位位置[1] := HMI.点位P5[1]; END_IF
IF _w11 THEN 定位位置[2] := HMI.点位P5[2]; END_IF
IF _w11 THEN 定位位置[3] := HMI.点位P5[3]; END_IF
所有轴启动 S= _w11;
_w12 := _w11 AND 轴运行完成;
轴运行完成 R= _w12;
所有轴启动 R= _w12;
避开扫描周期 S= _w12;
IF _w12 THEN 下一步 := 10; END_IF

// NETWORK 10: ......

// NETWORK 11: ......
// 网络注释

// NETWORK 12: ......
// 网络注释

// NETWORK 13: 组合轴运行
// 网络注释
LS_4AxisLine_0(
    Axis0 := Axis,
    Axis1 := Axis_1,
    Axis2 := Axis_2,
    Axis3 := Axis_3,
    Exec := 所有轴启动,
    Stop := NOT I_List.X1,
    EndPos := 定位位置,
    Velocity := 100,
    Acceleration := 100,
    Deceleration := 100); // LS_4AxisLine
轴运行完成 S= LS_4AxisLine_0.Done;

END_PROGRAM
